(* IEC 61131-3 sources: OSCAT_OpenPLC/OSCAT BUILDING 1.00/OSCAT BUILDING 1.0/build (part 3) *)

  (* From OSCAT Library, www.OSCAT.de *)
  (* T_PLC_MS, ONTIME required *)
END_FUNCTION_BLOCK

FUNCTION_BLOCK ACTUATOR_A
  VAR_INPUT
    I1 : BYTE;
    I2 : BYTE;
    IS : BOOL;
    RV : BOOL;
    DX : BOOL;
    RUNTIME : TIME;
    SELF_ACT_TIME : TIME;
    OUT_MIN : DWORD;
    OUT_MAX : DWORD;
  END_VAR
  VAR_OUTPUT
    Y : DWORD;
  END_VAR
  VAR
    timer : CYCLE_4;
    dx_edge : BOOL;
  END_VAR

  (* run the system timer, if self_act_time = t#0s then state is set to 0 *)
  timer(T0 := RUNTIME, T1 := RUNTIME, T3 := SELF_ACT_TIME, sl := DX AND NOT dx_edge, sx := 0, S0 := SELF_ACT_TIME > t#0s);
  dx_edge := dx;

  CASE timer.STATE OF
  	0: 	(* self act min value *)
  		Y := OUT_MIN;
  	1:	(* self_act max value *)
  		Y := OUT_MAX;
  	3:	(* normal operation *)
  		IF rv THEN
  			Y := UDINT_TO_DWORD(DWORD_TO_UDINT(OUT_MAX) - (DWORD_TO_UDINT(OUT_MAX) - DWORD_TO_UDINT(OUT_MIN)) * BYTE_TO_UDINT(SEL(IS, I1, I2)) / UDINT#255);
  		ELSE
  			Y := UDINT_TO_DWORD((DWORD_TO_UDINT(OUT_MAX) - DWORD_TO_UDINT(OUT_MIN)) * BYTE_TO_UDINT(SEL(IS, I1, I2)) / UDINT#255 + DWORD_TO_UDINT(OUT_MIN));
  		END_IF;
  END_CASE;

  (* From OSCAT Library, www.OSCAT.de *)
  (* Cycle_4 required *)
END_FUNCTION_BLOCK

FUNCTION_BLOCK BLIND_CONTROL
  VAR_INPUT
    UP : BOOL;
    DN : BOOL;
    S_IN : BYTE;
    PI : BYTE;
    AI : BYTE;
    T_UD : TIME;
    T_ANGLE : TIME;
    T_LOCKOUT : TIME := t#100ms;
    SENS : BYTE := 5;
  END_VAR
  VAR_OUTPUT
    POS : BYTE;
    ANG : BYTE;
    MU : BOOL;
    MD : BOOL;
    STATUS : BYTE;
  END_VAR
  VAR
    act : BLIND_ACTUATOR;
    delta : BYTE;
    ipos : BYTE;
    iangel : BYTE;
    bTimeTest : BOOL;
  END_VAR

  IF bTimeTest THEN
  	PI:=iPos;
  	AI:=iAngel;
  	UP:=TRUE;
  	DN:=TRUE;
  END_IF;

  (* Check Position*)
  act(T_UD:=T_UD, T_ANGLE:=T_ANGLE, T_lockout := T_Lockout);

  IF UP AND DN THEN
  	(* automatic modus detected *)
  	(* first find correct position *)
  	IF BYTE_TO_INT(act.pos) < BYTE_TO_INT(pi) - BYTE_TO_INT(delta) THEN
  		act.UP := TRUE;
  		act.DN := FALSE;
  		delta := BYTE#0;
  		STATUS := BYTE#121;
  	ELSIF BYTE_TO_INT(act.pos) > BYTE_TO_INT(pi) + BYTE_TO_INT(delta) THEN
  		act.UP := FALSE;
  		act.DN := TRUE;
  		delta := BYTE#0;
  		STATUS := BYTE#122;
  	(* regulate angle *)
  	ELSIF BYTE_TO_INT(act.ang) < BYTE_TO_INT(ai) - BYTE_TO_INT(delta) AND T_angle > T#100ms THEN
  		act.UP := TRUE;
  		act.DN := FALSE;
  		delta := SHR(sens,2);
  		STATUS := BYTE#123;
  	ELSIF BYTE_TO_INT(act.ang) > BYTE_TO_INT(ai) + BYTE_TO_INT(delta) AND T_angle > T#100ms THEN
  		act.UP := FALSE;
  		act.DN := TRUE;
  		delta := SHR(sens,2);
  		STATUS := BYTE#124;
  	(* correct position reached *)
  	ELSE
  		act.UP := FALSE;
  		act.DN := FALSE;
  		delta := sens;
  		STATUS := S_IN;
  	END_IF;
  ELSE
  	act.UP := UP;
  	act.DN := DN;
  	STATUS := S_IN;
  END_IF;

  (* blind control calls blind_actuator *)
  act(T_UD:=T_UD, T_ANGLE:=T_ANGLE, T_lockout := T_Lockout);
  pos := act.pos;
  ang := act.ang;
  MU := act.QU;
  md := act.QD;
  status := act.status;

  (* From OSCAT LIBRARY, www.oscat.de *)
  (* BLIND_ACTUATOR required *)
END_FUNCTION_BLOCK

FUNCTION_BLOCK BLIND_INPUT
  VAR_INPUT
    POS : BYTE;
    ANG : BYTE;
    S1 : BOOL;
    S2 : BOOL;
    IN : BOOL;
    PI : BYTE;
    AI : BYTE;
    SINGLE_SWITCH : BOOL;
    CLICK_EN : BOOL := TRUE;
    CLICK_TIME : TIME := t#500ms;
    MAX_RUNTIME : TIME := t#60s;
    MANUAL_TIMEOUT : TIME := t#1h;
    DEBOUNCE_TIME : TIME := t#20ms;
    DBL_CLK1 : BOOL := FALSE;
    DBL_POS1 : BYTE;
    DBL_ANG1 : BYTE;
    DBL_CLK2 : BOOL := FALSE;
    DBL_POS2 : BYTE := 255;
    DBL_ANG2 : BYTE := 255;
    D1_TOGGLE : BOOL := TRUE;
    D2_TOGGLE : BOOL := TRUE;
    MASTER_MODE : BOOL;
  END_VAR
  VAR_OUTPUT
    QU : BOOL := TRUE;
    QD : BOOL := TRUE;
    STATUS : BYTE;
    PO : BYTE := 255;
    AO : BYTE := 255;
    D1 : BOOL;
    D2 : BOOL;
  END_VAR
  VAR
    s1e : TOF;
    s2e : TOF;
    s1d : CLICK_MODE;
    s2d : CLICK_MODE;
    dir : BOOL;
    tx : TIME;
    last : TIME;
  END_VAR

  tx:= UDINT_TO_TIME(T_PLC_MS(en:=true));

  (* inputs S1 and S2 are debounced and then decoded for multiple clicks *)
  s1e(in := S1, pt := DEBOUNCE_TIME);
  s2e(in := S2, pt := DEBOUNCE_TIME);
  s1d(in := (s1e.Q AND NOT SINGLE_SWITCH) OR (s1e.Q AND SINGLE_SWITCH AND dir), t_long := CLICK_TIME);
  s2d(in := (s2e.Q AND NOT SINGLE_SWITCH) OR (s1e.Q AND SINGLE_SWITCH AND NOT dir), t_long := CLICK_TIME);

  (* if d1 and d2 are not toggle clear them to make sure they are only active for oine cycle *)
  IF NOT d1_toggle THEN d1 := FALSE; END_IF;
  IF NOT d2_toggle THEN d2 := FALSE; END_IF;

  (* decode actions *)
  IF (s1d.LONG AND s2d.LONG) OR (status = BYTE#139) THEN
     status := BYTE#139;
     IF NOT (s1d.LONG OR s2d.LONG)  THEN status := BYTE#130; END_IF;
  ELSIF s1d.tp_LONG THEN
  	status := BYTE#132;
  ELSIF s2d.tp_LONG THEN
  	status := BYTE#133;
  ELSIF  s1d.SINGLE THEN
  	IF click_en THEN
  		(* if running then we stop otherwise start new direction *)
  		IF QU XOR QD THEN
  			status := BYTE#131;
  		ELSE
  			status := BYTE#134;
  			last := tx;
  			dir := NOT dir;
  		END_IF;
  	END_IF;
  ELSIF  s2d.SINGLE THEN
  	IF click_en THEN
  		(* if running then we stop otherwise start new direction *)
  		IF QU XOR QD THEN
  			status := BYTE#131;
  		ELSE
  			status := BYTE#135;
  			last := tx;
  			dir := NOT dir;
  		END_IF;
  	END_IF;
  ELSIF in THEN
  	status := BYTE#136;
  	last := tx;
  ELSIF s1d.DOUBLE THEN
  	IF dbl_clk1 THEN
  		(* a position need to be set for a double click on S1 *)
  		status := BYTE#137;
  		last := tx;
  	ELSE
  		(* toggle the output when dbl_clk1 is not active *)
  		D1 := NOT D1;
  	END_IF;
  ELSIF s2d.DOUBLE THEN
  	IF dbl_clk2 THEN
  		(* a position need to be set for a double click on S2 *)
  		status := BYTE#138;
  		last := tx;
  	ELSE
  		(* toggle the output when dbl_clk2 is not active *)
  		(* in single switch mode we need to toggle d1 instead of d2 *)
  		IF single_switch THEN D1 := NOT D1; ELSE D2 := NOT D2; END_IF;
  	END_IF;
  END_IF;

  (* state machine *)
  CASE BYTE_TO_INT(status) OF
  	0:		(* power up operation *)
  			status := BYTE#130;

  	130:	(* automatic operation standby *)
  			IF NOT master_mode THEN
  				PO := POS;
  				AO := ANG;
  			END_IF;
  			QU := TRUE;
  			QD := TRUE;

  	131:	(* manual operation standby *)
  			QU := FALSE;
  			QD := FALSE;
  			PO := POS;
  			AO := ANG;
  			(* manual mode will be ended when timeout is reached *)
  			IF tx - last >= manual_timeout THEN
  				status := BYTE#130;
  			END_IF;

  	132:	(* manual operation up *)
  			QU := TRUE;
  			QD := FALSE;
  			PO := POS; AO := ANG;
  			last := tx;
  			IF NOT s1d.LONG THEN status := BYTE#131; dir := NOT dir; END_IF;

  	133:	(* manual operation down *)
  			QU := FALSE;
  			QD := TRUE;
  			PO := POS; AO := ANG;
  			last := tx;
  			IF NOT s2d.LONG THEN	status := BYTE#131; dir := NOT dir; END_IF;

  	134:	(* manual operation single click up *)
  			QU := TRUE;
  			QD := FALSE;
  			PO := POS; AO := ANG;
  			IF tx - last >= max_runtime THEN status := BYTE#131; END_IF;

  	135:	(* manual operation single click dn *)
  			QU := FALSE;
  			QD := TRUE;
  			PO := POS; AO := ANG;
  			IF tx - last >= max_runtime THEN status := BYTE#131;	END_IF;

  	136:	(* forced input in = true *)
  			QU := TRUE;
  			QD := TRUE;
  			PO := PI; AO := AI;
  			IF tx-last >= max_runtime THEN status := BYTE#130; END_IF;

  	137:	(* double click1 position *)
  			QU := TRUE;
  			QD := TRUE;
  			PO := DBL_POS1;
  			AO := DBL_ANG1;
  			IF tx - last >= max_runtime THEN status := BYTE#131; END_IF;

  	138:	(* double click2 position *)
  			QU := TRUE;
  			QD := TRUE;
  			PO := DBL_POS2;
  			AO := DBL_ANG2;
  			IF tx - last >= max_runtime THEN status := BYTE#131; END_IF;

  	   139:   (* manual operation standby *)
  	         QU := FALSE;
  	         QD := FALSE;
  	         PO := POS;
  	         AO := ANG;

  END_CASE;

  (* From OSCAT LIBRARY, www.oscat.de *)
  (* T_PLC_MS required *)
END_FUNCTION_BLOCK

FUNCTION_BLOCK SWITCH_I
  VAR_INPUT
    SET : BOOL;
    IN : BOOL;
    RST : BOOL;
    T_DEBOUNCE : TIME := t#10ms;
    T_RECONFIG : TIME := t#1s;
    T_ON_MAX : TIME := t#0h;
  END_VAR
  VAR_OUTPUT
    Q : BOOL := FALSE;
  END_VAR
  VAR
    state : BYTE := 0;
    edge : BOOL := FALSE;
    _r_edge : BOOL := FALSE;
    T_on : TIME;
    tx : TIME;
  END_VAR

  tx:= UDINT_TO_TIME(T_PLC_MS(en:=true));

  (* asynchronous set and reset first *)
  IF set AND NOT rst THEN
  	Q := TRUE;
  	T_on := tx;
  ELSIF rst THEN
  	Q := FALSE;
  (* check FOR input edge AND start debounce timer *)
  ELSIF (in XOR edge) AND NOT (state = BYTE#1) THEN
  	state := BYTE#1;
  	T_on := Tx;
  (* edge was detected and debounce time elapsed *)
  ELSIF (state = BYTE#1) AND (Tx - t_debounce >= T_on) THEN
  	state := BYTE#2;
  	(* react on rising or falling edge depending on r_edge *)
  	IF _r_edge XOR in THEN Q := NOT Q; END_IF;
  (* wait for T_reconfig and adjust r_edge *)
  ELSIF state = BYTE#2 AND Tx - t_reconfig >= T_on THEN
  	_r_edge := in;
  END_IF;
  IF Q AND T_on_max > t#0ms AND Tx >= T_on + T_on_max THEN
  	Q := FALSE;
  END_IF;
  edge := in;

  (* From OSCAT LIBRARY, www.oscat.de *)
END_FUNCTION_BLOCK

FUNCTION_BLOCK PULSE_T
  VAR_INPUT
    IN : BOOL;
    T1 : TIME;
    T2 : TIME;
    RST : BOOL;
  END_VAR
  VAR_OUTPUT
    Q : BOOL;
  END_VAR
  VAR
    init : BOOL;
    last : TIME;
    tx : TIME;
    edge : BOOL;
  END_VAR

  tx:= UDINT_TO_TIME(T_PLC_MS(en:=true));

  IF NOT init THEN
  	init := TRUE;
  	last := tx;
  ELSIF RST THEN
  	(* asynchronous reset *)
  	Q := FALSE;
  ELSIF IN AND NOT edge AND NOT Q THEN
  	(* a rising edge on in will reversre the output status, if new pulse is startet the start time is stored in last *)
  	last := tx;
  	Q := TRUE;
  ELSIF NOT IN AND edge AND ((tx - last) > T1) THEN
  	(* a falling edge on IN will clear the output if in was high for more then T1 *)
  	Q := FALSE;
  ELSIF (tx - last) >= T2 THEN
  	(* timeout for long pulse if second click did not occur or in stays high *)
  	Q := FALSE;
  END_IF;

  edge := IN;

  (* From OSCAT LIBRARY, www.oscat.de *)
  (* T_PLC_MS required *)
END_FUNCTION_BLOCK

FUNCTION AIR_ENTHALPY : REAL
  VAR_INPUT
    _T : REAL;
    RH : REAL;
  END_VAR

  Air_enthalpy := 1.00482 * _T + (1.86 * _T + 2500.78) * dew_con(RH,_T);

  (* From OSCAT Library, www.OSCAT.de *)
  (* DEW_CON required *)
END_FUNCTION

FUNCTION_BLOCK PULSE_LENGTH
  VAR_INPUT
    IN : BOOL;
    T_SHORT : TIME := t#100ms;
    T_LONG : TIME := t#1s;
  END_VAR
  VAR_OUTPUT
    SHORT : BOOL;
    MIDDLE : BOOL;
    LONG : BOOL;
  END_VAR
  VAR
    tx : TIME;
    tn : TIME;
    edge : BOOL;
  END_VAR

  tx:= UDINT_TO_TIME(T_PLC_MS(en:=true));

  (* reset outputs, they should only be active 1 cycle *)
  short := FALSE;
  Middle := FALSE;
  long := FALSE;

  (* detect rising edge *)
  IF in AND NOT edge THEN
  	edge := TRUE;
  	tn := tx;

  (* detect for falling edge *)
  ELSIF NOT in AND edge THEN
  	edge := FALSE;
  	tn := tx - tn;
  	IF tn < t_short THEN
  		short := TRUE;
  	ELSIF tn > t_long THEN
  		long := TRUE;
  	ELSE
  		Middle := TRUE;
  	END_IF;

  (* generate long pulse as soon as T_long is reached *)
  ELSIF in AND tx - tn > t_long THEN
  	long := TRUE;
  END_IF;

  (* From OSCAT LIBRARY, www.oscat.de *)
END_FUNCTION_BLOCK

FUNCTION_BLOCK SWITCH_X
  VAR_INPUT
    IN1 : BOOL;
    IN2 : BOOL;
    IN3 : BOOL;
    IN4 : BOOL;
    IN5 : BOOL;
    IN6 : BOOL;
    T_DEBOUNCE : TIME := t#50ms;
  END_VAR
  VAR_OUTPUT
    Q1 : BOOL;
    Q2 : BOOL;
    Q3 : BOOL;
    Q4 : BOOL;
    Q5 : BOOL;
    Q6 : BOOL;
    Q31 : BOOL;
    Q41 : BOOL;
    Q51 : BOOL;
    Q61 : BOOL;
    Q32 : BOOL;
    Q42 : BOOL;
    Q52 : BOOL;
    Q62 : BOOL;
  END_VAR
  VAR
    init : BOOL;
    T1 : TOF;
    T2 : TOF;
    T3 : TOF;
    T4 : TOF;
    T5 : TOF;
    T6 : TOF;
    tx : TIME;
    x1 : BOOL;
    x2 : BOOL;
    E1 : BOOL;
    E2 : BOOL;
  END_VAR

  (* initialize on startup *)
  IF NOT init THEN
  	init := TRUE;
  	IF t_debounce < t#50ms THEN tx := t#50ms; ELSE tx := t_debounce; END_IF;
  	T1(PT := Tx);
  	T2(PT := Tx);
  	T3(PT := Tx);
  	T4(PT := Tx);
  	T5(PT := Tx);
  	T6(PT := Tx);
  ELSE
  	Q1 := FALSE;
  	Q2 := FALSE;
  	Q3 := FALSE;
  	Q4 := FALSE;
  	Q5 := FALSE;
  	Q6 := FALSE;
  	Q31 := FALSE;
  	Q41 := FALSE;
  	Q51 := FALSE;
  	Q61 := FALSE;
  	Q32 := FALSE;
  	Q42 := FALSE;
  	Q52 := FALSE;
  	Q62 := FALSE;
  END_IF;

  (* read inputs and debounce *)
  	T1(IN := IN1);
  	T2(IN := IN2);
  	T3(IN := IN3);
  	T4(IN := IN4);
  	T5(IN := IN5);
  	T6(IN := IN6);

  (* detect edge of IN1 and IN2 *)
  IF t1.Q AND NOT E1 THEN X1 := TRUE; END_IF;
  IF t2.Q AND NOT E2 THEN X2 := TRUE; END_IF;

  IF t1.Q THEN
  	IF t3.q THEN
  		q31 := TRUE;
  		X1 := FALSE;
  	ELSIF t4.q THEN
  		q41 := TRUE;
  		X1 := FALSE;
  	ELSIF t5.q THEN
  		q51 := TRUE;
  		X1 := FALSE;
  	ELSIF t6.q THEN
  		q61 := TRUE;
  		X1 := FALSE;
  	END_IF;
  ELSIF t2.Q THEN
  	IF t3.q THEN
  		q32 := TRUE;
  		X2 := FALSE;
  	ELSIF t4.q THEN
  		q42 := TRUE;
  		X2 := FALSE;
  	ELSIF t5.q THEN
  		q52 := TRUE;
  		X2 := FALSE;
  	ELSIF t6.q THEN
  		q62 := TRUE;
  		X2 := FALSE;
  	END_IF;
  (* in1 was active alone *)
  ELSIF NOT T1.Q AND E1 AND X1 THEN
  	Q1 := TRUE;
  	X1 := FALSE;
  ELSIF NOT T2.Q AND E2 AND X2 THEN
  	Q2 := TRUE;
  	X2 := FALSE;
  ELSIF T3.Q THEN
  	Q3 := TRUE;
  ELSIF T4.Q THEN
  	Q4 := TRUE;
  ELSIF T5.Q THEN
  	Q5 := TRUE;
  ELSIF T6.Q THEN
  	Q6 := TRUE;
  END_IF;

  (* save state of in1 and in2 *)
  E1 := T1.Q;
  E2 := T2.Q;

  (* From OSCAT LIBRARY, www.oscat.de *)
END_FUNCTION_BLOCK

FUNCTION_BLOCK F_LAMP
  VAR_INPUT
    SWITCH : BOOL;
    DIMM : BYTE := 255;
    RST : BOOL;
    T_NO_DIMM : UINT := 100;
    T_MAINTENANCE : UINT := 15000;
  END_VAR
  VAR_OUTPUT
    LAMP : BYTE;
    STATUS : BYTE;
  END_VAR
  VAR_IN_OUT
    _ONTIME : UDINT;
    CYCLES : UDINT;
  END_VAR
  VAR
    runtime : ONTIME;
  END_VAR

  runtime(in := switch, SECONDS := _ONTIME , CYCLES := CYCLES);
  CYCLES := runtime.CYCLES;
  _ONTIME := runtime.SECONDS;

  IF RST THEN
  	_ONTIME := UDINT#0;
  	CYCLES := UDINT#0;
  END_IF;
  IF SWITCH THEN
  	IF _ontime < UINT_TO_UDINT(T_NO_DIMM) * UDINT#3600 THEN
  		LAMP := BYTE#255;
  		STATUS := BYTE#111;
  	ELSE
  		LAMP := DIMM;
  		STATUS := BYTE#112;
  	END_IF;
  ELSE
  	LAMP := BYTE#0;
  	STATUS := BYTE#110;
  END_IF;

  IF _ontime >= UINT_TO_UDINT(T_maintenance) * UDINT#3600 AND T_Maintenance > UINT#0 THEN
  	STATUS := BYTE#120;
  END_IF;

  (* From OSCAT LIBRARY, www.oscat.de *)
  (* ONTIME required *)
END_FUNCTION_BLOCK

FUNCTION TANK_VOL2 : REAL
  VAR_INPUT
    TR : REAL;
    H : REAL;
  END_VAR

  TANK_VOL2 := 3.14159265358979323846264338327950288 * H * H * (TR - H / 3.0);

  (* From OSCAT Library, www.OSCAT.de *)
END_FUNCTION

FUNCTION TANK_VOL1 : REAL
  VAR_INPUT
    TR : REAL;
    TL : REAL;
    H : REAL;
  END_VAR

  TANK_VOL1 := CIRCLE_SEG(TR, H) * TL;

  (* From OSCAT Library, www.OSCAT.de *)
  (* CIRCLE_SEG required *)
END_FUNCTION

FUNCTION DT_TO_TOD_2 : UDINT
  VAR_INPUT
    IN : UDINT;
  END_VAR

  DT_TO_TOD_2 := (IN MOD UDINT#86400) * UDINT#1000;

  (* From OSCAT Library, www.oscat.de *)
END_FUNCTION

FUNCTION_BLOCK ACTUATOR_UD
  VAR_INPUT
    UD : BOOL;
    _ON : BOOL;
    MANUAL : BOOL;
    UP : BOOL;
    DN : BOOL;
    OFF : BOOL;
    YUP_IN : BOOL;
    YDN_IN : BOOL;
    OUT_RETURN : BOOL;
    _TON : TIME;
    _TOFF : TIME;
  END_VAR
  VAR_OUTPUT
    YUP : BOOL;
    YDN : BOOL;
    STATUS : BYTE;
  END_VAR
  VAR
    tx : TIME;
    last : TIME;
    init : BOOL;
  END_VAR

  tx:= UDINT_TO_TIME(T_PLC_MS(en:=true));

  IF NOT init THEN
  	(* INITIALIZATION AT FIRST CALL *)
  	last := tx;
  	init := TRUE;
  ELSIF off THEN
  	(* emergency shut off detected *)
  	Yup := FALSE;
  	Ydn := FALSE;
  	last := tx;
  	status := BYTE#101;

  (* WATH FOR MIN TON TIME *)
  ELSIF ((Yup OR Ydn) AND tx - last < _Ton) THEN RETURN;
  ELSIF NOT yup AND NOT ydn AND tx - last < _toff THEN	RETURN;

  (* manual operation *)
  ELSIF manual THEN
  	status := BYTE#102;
  	(* directional chage set both outs 0 first *)
  	IF yup AND NOT up OR ydn AND NOT dn THEN
  		ydn := FALSE;
  		yup := FALSE;
  		last := tx;
  	(* manual up operation *)
  	ELSIF UP AND NOT DN AND NOT OFF THEN
  		Ydn := FALSE;
  		Yup := TRUE;
  		last := tx;
  		status := BYTE#103;
  	(* manual down operation *)
  	ELSIF DN AND NOT UP AND NOT OFF THEN
  		Yup := FALSE;
  		Ydn := TRUE;
  		last := tx;
  		status := BYTE#104;
  	(* maual mode but no up or down *)
  	ELSE
  		IF YUP OR YDN THEN LAST := tx; END_IF;
  		Yup := FALSE;
  		Ydn := FALSE;
  	END_IF;

  (* automatic operation *)
  ELSE
  	(* directional change set outputs low first *)
  	IF yup AND NOT ud OR ydn AND UD THEN
  		yup := FALSE;
  		ydn := FALSE;
  		last := tx;
  	(* automatic up operation *)
  	ELSIF Ud AND _on AND NOT OFF THEN
  		Ydn := FALSE;
  		Yup := TRUE;
  		last := tx;
  		status := BYTE#111;

  	(* automatic down operation *)
  	ELSIF NOT UD AND _on AND NOT OFF THEN
  		Yup := FALSE;
  		Ydn := TRUE;
  		last := tx;
  		status := BYTE#112;
  	(* standby mode *)
  	ELSE
  		IF Yup OR Ydn THEN last := tx; END_IF;
  		Yup := FALSE;
  		Ydn := FALSE;
  		status := BYTE#110;
  	END_IF;
  END_IF;

  (* make sure Yup and Ydn are never on at the same time *)
  IF Ydn AND Yup_in AND out_return THEN
  	Ydn := FALSE;
  	status := BYTE#1;
  END_IF;
  IF Yup AND Ydn_in AND out_return THEN
  	Yup := FALSE;
  	status := BYTE#2;
  END_IF;

  (* From OSCAT Library, www.OSCAT.de *)
  (* T_PLC_MS required *)
END_FUNCTION_BLOCK

FUNCTION_BLOCK ACTUATOR_3P
  VAR_INPUT
    IN : BYTE;
    TEST : BOOL;
    ARE : BOOL := TRUE;
    END_POS : BOOL;
    T_RUN : TIME := t#60s;
    T_EXT : TIME := t#10s;
    T_CAL : TIME := t#600s;
    T_DIAG : TIME := t#10d;
    SWITCH_AVAIL : BOOL;
  END_VAR
  VAR_OUTPUT
    OUT1 : BOOL;
    OUT2 : BOOL;
    POS : BYTE;
    ERROR : BOOL;
    STATUS : BYTE;
  END_VAR
  VAR_IN_OUT
    ARX : BOOL;
  END_VAR
  VAR
    tx : TIME;
    _ramp : _RMP_NEXT;
    next_cal : TIME;
    next_diag : TIME;
    last : TIME;
    start : TIME;
  END_VAR

  tx := UDINT_TO_TIME(T_PLC_MS(en:=true));

  (* check test input *)
  IF TEST THEN
  	status := BYTE#103;
  	start := tx;
  	ARX := TRUE;
  END_IF;

  CASE BYTE_TO_INT(status) OF
  	0:	(* power on setup *)
  		IF ARE AND NOT ARX THEN
  			status := BYTE#103;
  			start := tx;
  			ARX := TRUE;
  		END_IF;

  	100:	(* normal operation *)
  		(* check for auto diagnostics *)
  		IF T_DIAG > T#0s AND tx > next_diag AND ARE AND NOT ARX THEN
  				status := BYTE#103;
  				start := tx;
  				ARX := TRUE;

  		(* check for auto calibration *)
  		ELSIF T_CAL > T#0s AND tx > next_cal AND ARE AND NOT ARX THEN
  			IF pos > BYTE#127 THEN
  				OUT1 := TRUE;
  				OUT2 := FALSE;
  				_ramp.IN := BYTE#255;
  				ARX := TRUE;
  			ELSE
  				OUT1 := FALSE;
  				OUT2 := TRUE;
  				_ramp.IN := BYTE#0;
  				ARX := TRUE;
  			END_IF;
  			status := BYTE#101;
  			start := tx;
  		ELSE
  			(* increment next_cal if not active *)
  			IF NOT(OUT1 OR OUT2) THEN next_cal := next_cal + (tx-last); END_IF;
  			(* set ramp generator to IN *)
  			_ramp.IN := IN;
  		END_IF;

  	101:	(* calibrate *)
  		IF tx - start < T_EXT THEN
  			next_cal := tx + T_CAL;
  		ELSIF SWITCH_AVAIL AND END_POS THEN
  			STATUS := BYTE#100;
  			ARX := FALSE;
  		ELSIF tx - start > T_EXT + T_RUN THEN
  			ERROR := SWITCH_AVAIL;
  			ARX := FALSE;
  		END_IF;

  	103:	(* diagnostics up*)
  		(* run up for T_ext *)
  		IF tx - start < T_EXT THEN
  			ERROR := FALSE;
  			_ramp.TR := T_RUN;
  			_ramp.TF := T_RUN;
  			OUT1 := TRUE;
  			OUT2 := FALSE;
  			_ramp.IN := BYTE#255;
  		ELSIF SWITCH_AVAIL AND END_POS THEN
  			_ramp.TR := tx - start;
  			STATUS := BYTE#104;
  		ELSIF tx - start > T_EXT + T_RUN THEN
  			ERROR := SWITCH_AVAIL;
  			STATUS := BYTE#104;
  			start := tx;
  		END_IF;

  	104:	(* diagnostics dn*)
  		IF tx - start < T_ext THEN
  			OUT1 := FALSE;
  			OUT2 := TRUE;
  			_ramp.IN := BYTE#0;
  			next_diag := tx + T_DIAG;
  		ELSIF SWITCH_AVAIL AND END_POS THEN
  			_ramp.TR := tx - start;
  			(* check if runtimes differ by more than 10% *)
  			IF DINT_TO_TIME(ABS(TIME_TO_DINT(_ramp.TR) - TIME_TO_DINT(_ramp.TF)) * DINT#10) > T_RUN THEN error := TRUE; END_IF;
  			STATUS := BYTE#100;
  			ARX := FALSE;
  			next_cal := tx + T_CAL;
  		ELSIF tx - start > T_EXT + T_RUN THEN
  			IF SWITCH_AVAIL THEN ERROR := TRUE; END_IF;
  			STATUS := BYTE#100;
  			ARX := FALSE;
  			next_CAL := tx + T_CAL;
  		END_IF;
  END_CASE;

  (* internal flap simulation and output activation *)
  _ramp(OUT := POS);
  POS := _ramp.OUT;
  IF STATUS = BYTE#100 THEN
  	OUT1 := _ramp.UP;
  	OUT2 := _ramp.DN;
  END_IF;

  (* adjust position if end switch is active *)
  IF SWITCH_AVAIL AND END_POS THEN
  	POS := SEL(POS > BYTE#127, BYTE#0, BYTE#255);
  	next_cal := tx + T_CAL;
  END_IF;

  (* set last to tx for next cycle *)
  last := tx;

  (* From OSCAT Library, www.OSCAT.de *)
  (* _RMP_NEXT required *)
END_FUNCTION_BLOCK

PROGRAM program0
  VAR
    LocalVar0 : DINT;
    LocalVar1 : DINT;
    LocalVar2 : DINT;
    ADD1_OUT : DINT;
  END_VAR

  ADD1_OUT := ADD(LocalVar0, LocalVar1);
  LocalVar2 := ADD1_OUT;
END_PROGRAM

FUNCTION_BLOCK FILTER_I
  VAR_INPUT
    X : INT;
    _T : TIME;
  END_VAR
  VAR_OUTPUT
    Y : INT;
  END_VAR
  VAR
    Yi : DINT;
    last : UDINT;
    tx : UDINT;
    init : BOOL;
  END_VAR

  tx:= T_PLC_MS(en:=true);

  (* startup initialisation *)
  IF NOT init OR _T = t#0s THEN
  	init := TRUE;
  	Yi := INT_TO_DINT(X) * DINT#1000;
  ELSE
  	(* to increase accuracy of the filter we calculate internal Yi wich is Y * 1000 *)
  	Yi := Yi + INT_TO_DINT(X - Y) * UDINT_TO_DINT(tx - last) * DINT#1000 / TIME_TO_DINT(_T);
  END_IF;
  last := tx;
  Y := DINT_TO_INT(yi / DINT#1000);

  (* From OSCAT Library, www.oscat.de *)
  (* T_PLC_MS required *)
END_FUNCTION_BLOCK

FUNCTION INC1 : INT
  VAR_INPUT
    X : INT;
    N : INT;
  END_VAR

  IF X >= N - 1 THEN
  	INC1 := 0;
  ELSE
  	INC1 := X + 1;
  END_IF;
  (* from OSCAT library; www.oscat.de  *)
END_FUNCTION

FUNCTION WCT : REAL
  VAR_INPUT
    _T : REAL;
    V : REAL;
  END_VAR

  IF V < 5.0 OR _T > 10.0 THEN
  	WCT := _T;
  ELSE
  	WCT := 13.12 + 0.6215 * _T +(0.3965 * _T - 11.37) * EXP(LN(v) * 0.16);
  END_IF;

  (* From OSCAT LIBRARY, www.oscat.de *)
END_FUNCTION

FUNCTION_BLOCK HEAT_TEMP
  VAR_INPUT
    T_EXT : REAL;
    T_INT : REAL;
    OFFSET : REAL;
    T_REQ : REAL;
    TY_MAX : REAL := 70.0;
    TY_MIN : REAL := 25.0;
    TY_CONFIG : REAL := 70.0;
    T_INT_CONFIG : REAL := 20.0;
    T_EXT_CONFIG : REAL := -15.0;
    T_DIFF : REAL := 10.0;
    C : REAL := 1.33;
    H : REAL := 3.0;
  END_VAR
  VAR_OUTPUT
    TY : REAL;
    HEAT : BOOL;
  END_VAR
  VAR
    tr : REAL;
    tx : REAL;
  END_VAR

  tr := T_INT + OFFSET;
  tx := (tr - T_EXT) / (T_INT_CONFIG - T_EXT_CONFIG);

  IF T_EXT + H > tr THEN
  	TY := 0.0;
  ELSE
  	TY := LIMIT(TY_MIN, tr + T_DIFF * 0.5 * tx + (TY_CONFIG - T_DIFF * 0.5 - tr) * EXPT(tx, 1.0 / C), TY_MAX);
  END_IF;

  TY := MAX(TY, T_REQ);
  HEAT := TY > 0.0;

  (* from OSCAT library www.oscat.de *)
END_FUNCTION_BLOCK

FUNCTION_BLOCK GEN_PULSE
  VAR_INPUT
    ENQ : BOOL := TRUE;
    PTH : TIME;
    PTL : TIME;
  END_VAR
  VAR_OUTPUT
    Q : BOOL;
  END_VAR
  VAR
    tx : TIME;
    tn : TIME;
    init : BOOL;
  END_VAR

  IF enq THEN
  		tx:= UDINT_TO_TIME(T_PLC_MS(en:=true));
  	IF NOT init THEN init := TRUE; tn := tx; END_IF;
  	IF tx - tn >= SEL(Q, PTL, PTH) THEN
  		tn := tn + SEL(Q, PTL, PTH);
  		Q := NOT Q;
  	END_IF;
  ELSE
  	Q := FALSE;
  	init := FALSE;
  END_IF;

  (* From OSCAT Library, www.OSCAT.de *)
  (* T_PLC_MS required*)
END_FUNCTION_BLOCK

FUNCTION_BLOCK ACTUATOR_2P
  VAR_INPUT
    IN : BYTE;
    TEST : BOOL;
    ARE : BOOL := TRUE;
    CYCLE_TIME : TIME;
    SENS : BYTE;
    SELF_ACT_TIME : TIME;
    SELF_ACT_PULSE : TIME;
    SELF_ACT_CYCLES : INT := 1;
  END_VAR
  VAR_OUTPUT
    OUT : BOOL;
    ARO : BOOL;
  END_VAR
  VAR_IN_OUT
    ARX : BOOL;
  END_VAR
  VAR
    timer : AUTORUN;
    pwgen : GEN_PULSE;
  END_VAR

  (* run the autorun timer *)
  timer(trun := SELF_ACT_PULSE * (2 * SELF_ACT_CYCLES), toff := SELF_ACT_TIME, Test := TEST, ARE := ARE, arx := ARX);
  ARO := timer.ARO;

  (* run the pulse width generator *)
  IF aro THEN
  	pwgen(PTL := SELF_ACT_PULSE, PTH := SELF_ACT_PULSE);
  	out := pwgen.Q;
  ELSIF in < sens THEN
  	out := FALSE;
  ELSIF BYTE_TO_USINT(in) > USINT#255 - BYTE_TO_USINT(sens) THEN
  	out := TRUE;
  ELSE
  	pwgen.PTH := udint_to_time((time_to_udint(CYCLE_TIME) * BYTE_TO_udint(BAND_B(IN,SENS))  ) / BYTE_TO_udint(BYTE#255));
  	pwgen.PTL := CYCLE_TIME - pwgen.PTH;
  	pwgen();
  	out := pwgen.Q;
  END_IF;

  (* From OSCAT Library, www.OSCAT.de *)
  (* AUTORUN, GEN_PULE, BAND_B required *)
END_FUNCTION_BLOCK

FUNCTION SDD_NH3 : REAL
  VAR_INPUT
    _T : REAL;
  END_VAR

  IF _T < -33.65 THEN
  	SDD_NH3 := EXP(7.3396511649 - ( 1166.7498002 / ( _T + 192.37 )));
  ELSE
  	SDD_NH3 := EXP(11.210964456 - ( 2564.9140075 / ( _T + 262.741 )));
  END_IF;

  (* From OSCAT Library, www.OSCAT.de *)
END_FUNCTION

FUNCTION_BLOCK TEMP_EXT
  VAR_INPUT
    T_EXT1 : REAL;
    T_EXT2 : REAL;
    T_EXT3 : REAL;
    T_EXT_CONFIG : BYTE := 0;
    DT_IN : UDINT;
    T_EXT_MIN : REAL := -40.0;
    T_EXT_MAX : REAL := 60.0;
    T_EXT_DEFAULT : REAL := -10.0;
    HEAT_PERIOD_START : UDINT := 20995200;
    HEAT_PERIOD_STOP : UDINT := 10281600;
    COOL_PERIOD_START : UDINT := 07776000;
    COOL_PERIOD_STOP : UDINT := 23500800;
    HEAT_START_TEMP_DAY : REAL := 15.0;
    HEAT_START_TEMP_NIGHT : REAL := 10.0;
    HEAT_STOP_TEMP : REAL := 18.0;
    COOL_START_TEMP_DAY : REAL := 26.0;
    COOL_START_TEMP_NIGHT : REAL := 26.0;
    COOL_STOP_TEMP : REAL := 24.0;
    START_DAY : UDINT := 32400000;
    START_NIGHT : UDINT := 75600000;
    CYCLE_TIME : TIME := t#10m;
  END_VAR
  VAR_OUTPUT
    T_EXT : REAL;
    HEAT : BOOL;
    COOL : BOOL;
  END_VAR
  VAR
    tx : TIME;
    last_run : TIME;
    init : BOOL;
    cool_start : UDINT;
    cool_stop : UDINT;
    heat_start : UDINT;
    heat_stop : UDINT;
    xdate : UDINT;
    day : BOOL;
  END_VAR

  IF NOT init THEN
  	init := TRUE;
  	heat_start := SET_DATE(1972,MONTH_OF_DATE(heat_period_start),DAY_OF_MONTH(heat_period_start));
  	heat_stop := SET_DATE(1972,MONTH_OF_DATE(heat_period_stop),DAY_OF_MONTH(heat_period_stop));
  	cool_start := SET_DATE(1972,MONTH_OF_DATE(cool_period_start),DAY_OF_MONTH(cool_period_start));
  	cool_stop := SET_DATE(1972,MONTH_OF_DATE(cool_period_stop),DAY_OF_MONTH(cool_period_stop));
  END_IF;

  (* read system time *)
  tx:= UDINT_TO_TIME(T_PLC_MS(en:=true));

  (* for efficiency exit isf this program has been executed less then 1min ago *)
  IF tx - last_run < cycle_time THEN RETURN; END_IF;

  (* calculate frequently used variables *)
  xdate := SET_DATE(1972,MONTH_OF_DATE(DT_TO_DATE_2(dt_in)),DAY_OF_MONTH(DT_TO_DATE_2(dt_in)));
  day := DT_TO_TOD_2(dt_in) >= start_day AND  DT_TO_TOD_2(dt_in) < start_night;

  (* read the correct external temperature depending on the t_ext_config setting *)
  t_ext := MULTI_IN(t_ext1, t_ext2, t_ext3, t_ext_default, t_ext_min, t_ext_max, t_ext_config);

  (* dtermine heating *)
  IF (heat_start <= heat_stop AND xdate >= heat_start AND xdate <= heat_stop) OR (heat_start > heat_stop AND (xdate >= heat_start OR xdate <= heat_stop)) THEN
  	(* heating period id true check for temperature *)
  	IF day AND t_ext <= heat_start_temp_day THEN
  		heat := TRUE;
  	ELSIF NOT day AND t_ext <= heat_start_temp_night THEN
  		heat := TRUE;
  	ELSIF t_ext >= heat_stop_temp THEN
  		heat := FALSE;
  	END_IF;
  ELSE
  	heat := FALSE;
  END_IF;

  (* dtermine cooling *)
  IF (cool_start <= cool_stop AND xdate >= cool_start AND xdate <= cool_stop) OR (cool_start > cool_stop AND (xdate >= cool_start OR xdate <= cool_stop)) THEN
  	(* cooling period is true check for temperature *)
  	IF day AND t_ext >= cool_start_temp_day THEN
  		cool := TRUE;
  	ELSIF NOT day AND t_ext >= cool_start_temp_night THEN
  		cool := TRUE;
  	ELSIF t_ext <= cool_stop_temp THEN
  		cool := FALSE;
  	END_IF;
  ELSE
  	cool := FALSE;
  END_IF;

  last_run := tx;

  (* From OSCAT LIBRARY, www.oscat.de *)
  (* many FB's required :-)  *)
END_FUNCTION_BLOCK

CONFIGURATION Config0

  RESOURCE Res0 ON PLC
    TASK task0(INTERVAL := T#20ms,PRIORITY := 0);
    PROGRAM instance0 WITH task0 : program0;
  END_RESOURCE
END_CONFIGURATION
